Staubli VAL3: calcTool4p7En.dtx

bool bAbort = true
num nLangSet = 100
num nS1[4]
num nS2[4]
num nS3[4]
num nS4[4]
num nScX
num nScY
num nScZ
num nToolX = 192.690167
num nToolY = -28.471807
num nToolZ = 149.691768
num nXPosButTxt[9]
  [2] = 5
  [3] = 10
  [4] = 15
  [5] = 20
  [6] = 25
  [7] = 30
  [8] = 35
num nYPosButTxt = 13
pointRx pTempS[5]
  [0] = {fatherId=world[0]}
  [1] = {x=378.320625, y=240.768097, z=466.569838, rx=-127.167365, ry=20.154779, rz=59.793558, shoulder=lefty, elbow=epositive, wrist=wpositive, fatherId=world[0]}
  [2] = {x=378.320625, y=240.768097, z=466.569838, rx=-127.167365, ry=20.154779, rz=59.793558, shoulder=lefty, elbow=epositive, wrist=wpositive, fatherId=world[0]}
  [3] = {x=378.320625, y=240.768097, z=466.569838, rx=-127.167365, ry=20.154779, rz=59.793558, shoulder=lefty, elbow=epositive, wrist=wpositive, fatherId=world[0]}
  [4] = {x=378.320625, y=240.768097, z=466.569838, rx=-127.167365, ry=20.154779, rz=59.793558, shoulder=lefty, elbow=epositive, wrist=wpositive, fatherId=world[0]}
string sUsrMess[140]
  [0] = "Please select a Language"
  [1] = "Programm zur Toolberechnung"
  [2] = "Dieses Prog. errechnet anhand 4 POINTS,"
  [3] = "die kugelfoermig um einen gemeinsamen"
  [4] = "Mittelpkt angeordnet sind,die X, Y und"
  [5] = "Z-Werte des akt. Tools. Diese Points"
  [6] = "muessen geometrisch unabhaengig sein."
  [7] = "D.h. sie duerfen nicht in EINER"
  [8] = "gemeinsamen Ebene liegen !!!"
  [9] = "Teachen der Locations !"
  [10] = "Punkt aufnehmen "
  [11] = "Aufnahme des "
  [12] = ".Punkts"
  [13] = "-Here- druecken um Punkt zu speichern"
  [14] = "ABBRUCH"
  [15] = "VORGANG ABGEBROCHEN !!!"
  [16] = ".Punkt aufgenommen !!!"
  [17] = "Mitte"
  [18] = "gemittelt"
  [19] = "Gemitteltes Tool sofort setzten ?"
  [20] = "TOOL NICHT GESETZT !!!"
  [21] = "TOOL GESETZT !!!"
  [22] = "Abbrechen       "
  [23] = "Wollen Sie fortfahren ? "
  [24] = " JA"
  [25] = "NEIN"
  [26] = "Here"
  [27] = "Ergebnis der Toolberechnung"
  [28] = "Tool-X"
  [29] = "Tool-Y"
  [30] = "Tool-Z"
  [31] = "Gemitteltes Tool => TRSF user_tool"
  [32] = "Division durch 0 nicht moeglich !!!"
  [101] = "Program for ToolCalculation"
  [102] = "Program to calculate the Center of a"
  [103] = "Sphere thoughout 4 POINTS which are"
  [104] = "on the surface of his Sphere. The X-,"
  [105] = "Y- and Z-Toolval. will be calcutated."
  [106] = "These POINTS have to be geometricly"
  [107] = "independant=>POINTS don't have to be"
  [108] = "located in ONE plane!!!"
  [109] = "Teaching of Locations !"
  [110] = "Teaching Location"
  [111] = "Teaching of "
  [112] = ".Point"
  [113] = "To teach the Point press - Here -"
  [114] = "ABORT"
  [115] = "PROGRAM ABORTED !!!"
  [116] = ".Point teached !!!"
  [117] = "Center"
  [118] = "average"
  [119] = "Do you want to SET average Tool now ?"
  [120] = "TOOL NOT SET !!!"
  [121] = "TOOL SET !!!"
  [122] = "Abort"
  [123] = "Do you want to continue ?"
  [124] = "YES"
  [125] = " NO"
  [126] = "Here"
  [127] = "Result of the Toolcalculation"
  [128] = "Tool-X"
  [129] = "Tool-Y"
  [130] = "Tool-Z"
  [131] = "Average Tool => TRSF user_tool"
  [132] = "Division though 0 is not possible !!!"
trsf trCenter
trsf trSphere[4]
trsf trTempTool[4]
public trsf trUserTool
